// TIA Portal V20 export
DATA_BLOCK "ControlNodes"   // DB152
// stored: MemoryReserve 100, Namespace Unit1.Em11
   VAR
      em : "LAF_typeEmControlNode";
      emstate { S7_SetPoint := 'True'} : "LUC_typeStates";
      citiMap : Struct
         PMC : "LER_PMC_Input_Data";
         FlexNet { S7_SetPoint := 'True'} : "LER_FlexNet_Data";
      END_STRUCT;
      weightCheck : "Unit1.Em11.typeSequenceControlNode";
      emData : "LER_typePartData";
      SpecialFunctionMode : Struct
         DryRun : Struct
            JRdetectPV : Array[0..15] of Bool;
         END_STRUCT;
      END_STRUCT;
      cmWeightCheckJRDetect : "LBC_typeDigitalSignalControlNode";
      cmWeightCheckControl : "LER_WeightCheckControlNode";
      "=====미사용=====" { ExternalAccessible := 'False'; ExternalVisible := 'False'; ExternalWritable := 'False'} : Bool;
      cmWeightCheckStageLifUpDown : "LBC_typeTwoWayActuatorControlNode";
   END_VAR
BEGIN
END_DATA_BLOCK
